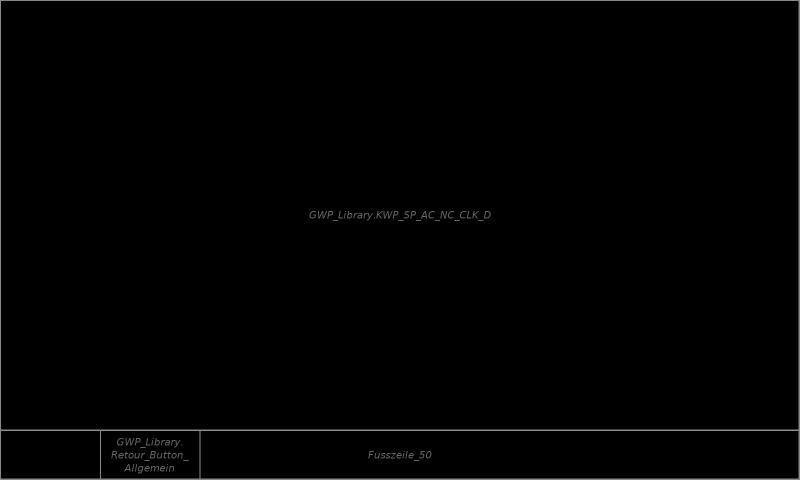
VISUALIZATION KWP_SP_AC_NC_CLK_D  // 800x480
    Frame (0,0 800x430)
        shows GWP_Library.KWP_SP_AC_NC_CLK_D(FB_CLK_D := Main.KWP_SP_AC_NC_0.GR_4_ohne_RE_0.TagNacht)
    Frame (0,430 800x50)
        shows Fusszeile_50()
    Frame (100,430 100x50)
        shows GWP_Library.Retour_Button_Allgemein()
END_VISUALIZATION

(* stored: Version 1.1.0.1, ProductVersion 3.1.4022.6
   Visu KWP_SP_AC_NC_CLK_D: Id {7ec31a02-cf49-4d36-888e-c94f8974e78a} *)
